// TIA Portal V20 export
ORGANIZATION_BLOCK "Startup"   // OB1005, LAD, Startup
TITLE = "Complete Restart"
// stored: AutoNumber false, Namespace Unit1.Em0, SetENOAutomatically false
   VAR_INPUT
      LostRetentive : Bool;   // True if retentive data are lost
      LostRTC : Bool;   // True if date and time are lost
   END_VAR
BEGIN

REGION Network 1 (SCL): Build the Absolut Reference Designator
   // Set the Absoult Reference Designator in the Config DB
   IF LEN(IN := "Unit1.Em0.Config".em.referenceDesignator.parent) <> 0 THEN
       "Unit1.Em0.Config".em.referenceDesignator.combined := CONCAT_WSTRING(IN1 := "Unit1.Em0.Config".em.referenceDesignator.parent, IN2 := WSTRING#'.', IN3 := "Unit1.Em0.Config".em.referenceDesignator.relative);
   ELSE
       "Unit1.Em0.Config".em.referenceDesignator.combined := "Unit1.Em0.Config".em.referenceDesignator.relative;
   END_IF;
END_REGION

REGION Network 2 (SCL): EM Startup
   "Unit1.Em0.HmiInterface".em.interlinkMode.isLinked := FALSE;
END_REGION

REGION Network 3 (SCL): Assign axes data
   // Assign axes
   "Unit1.Em0.Config".axis[1] := "BA010AZCRDR1_UnwinderLeftAxisB";

   // HW_SubModule
   "Unit1.Em0.Config".moduleAccessPoint[1] := "BA010AZCRCU1~BA010AZCRCU1_X150~BA010AZCRDR1_ModuleAccessPoint";
END_REGION

REGION Network 4 (SCL): EM Startup
   "Unit1.Em0.HmiInterface".em.interlinkMode.isLinked := FALSE;

   // FB Enable
   "Unit1.Em0.HmiInterface".cmUnWinderAxisB.commands.enable := TRUE;
END_REGION

REGION Network 5 (SCL): CM Config
   // Unwinder Axis B
   "Unit1.Em0.Config".cmUnWinderAxisB.referenceDesignator := WSTRING#'Left UnWinder Axis B';
   "Unit1.Em0.Config".cmUnWinderAxisB.disableAlarms := FALSE;
   "Unit1.Em0.Config".cmUnWinderAxisB.masterControlPopUp := TRUE;


   // Air Shaft
   "Unit1.Em0.Config".cmAirShaftOnOff.referenceDesignator := WSTRING#'Left Air Shaft';
   "Unit1.Em0.Config".cmAirShaftOnOff.monitoringLeavingFeedback := T#0MS;
   "Unit1.Em0.Config".cmAirShaftOnOff.monitoringReachingFeedback := T#0MS;
   "Unit1.Em0.Config".cmAirShaftOnOff.monitoringDiscrepancy := T#0ms;
   "Unit1.Em0.Config".cmAirShaftOnOff.setOutputHomeContinuously := TRUE;
   "Unit1.Em0.Config".cmAirShaftOnOff.setOutputWorkContinuously := TRUE;
   "Unit1.Em0.Config".cmAirShaftOnOff.disableHomeCommand := FALSE;
   "Unit1.Em0.Config".cmAirShaftOnOff.disableFeedbackHomePos := TRUE;
   "Unit1.Em0.Config".cmAirShaftOnOff.disableFeedbackWorkPos := TRUE;
   "Unit1.Em0.Config".cmAirShaftOnOff.disableAlarms := FALSE;
   "Unit1.Em0.Config".cmAirShaftOnOff.resetOutputsOnError := FALSE;
   "Unit1.Em0.Config".cmAirShaftOnOff.allwaysWaitOnReachingTime := FALSE;


   // Electrode Expel
   "Unit1.Em0.Config".cmExpelFwdBwd.referenceDesignator := WSTRING#'Left Electrode Expel';
   "Unit1.Em0.Config".cmExpelFwdBwd.monitoringLeavingFeedback := T#5s;
   "Unit1.Em0.Config".cmExpelFwdBwd.monitoringReachingFeedback := T#5s;
   "Unit1.Em0.Config".cmExpelFwdBwd.monitoringDiscrepancy := T#0ms;
   "Unit1.Em0.Config".cmExpelFwdBwd.setOutputHomeContinuously := TRUE;
   "Unit1.Em0.Config".cmExpelFwdBwd.setOutputWorkContinuously := TRUE;
   "Unit1.Em0.Config".cmExpelFwdBwd.disableHomeCommand := FALSE;
   "Unit1.Em0.Config".cmExpelFwdBwd.disableFeedbackHomePos := FALSE;
   "Unit1.Em0.Config".cmExpelFwdBwd.disableFeedbackWorkPos := FALSE;
   "Unit1.Em0.Config".cmExpelFwdBwd.disableAlarms := FALSE;
   "Unit1.Em0.Config".cmExpelFwdBwd.resetOutputsOnError := FALSE;
   "Unit1.Em0.Config".cmExpelFwdBwd.allwaysWaitOnReachingTime := FALSE;


   // Radius Measure
   "Unit1.Em0.Config".cmRadiusMeasureAnalogInput.referenceDesignator := WSTRING#'Left Radius Measure';
   "Unit1.Em0.Config".cmRadiusMeasureAnalogInput.physicalUnit := 'mm';
   "Unit1.Em0.Config".cmRadiusMeasureAnalogInput.isUnipolarSignal := TRUE;
   "Unit1.Em0.Config".cmRadiusMeasureAnalogInput.default := 0;
   "Unit1.Em0.Config".cmRadiusMeasureAnalogInput.limitHigh2 := 10000;
   "Unit1.Em0.Config".cmRadiusMeasureAnalogInput.limitHigh1 := 9000;
   "Unit1.Em0.Config".cmRadiusMeasureAnalogInput.limitLow1 := 40;
   "Unit1.Em0.Config".cmRadiusMeasureAnalogInput.limitLow2 := 30;
   "Unit1.Em0.Config".cmRadiusMeasureAnalogInput.processValueMax := 10000;
   "Unit1.Em0.Config".cmRadiusMeasureAnalogInput.processValueMin := 10;
   "Unit1.Em0.Config".cmRadiusMeasureAnalogInput.scaleAnalogUppPoint := 27648;
   "Unit1.Em0.Config".cmRadiusMeasureAnalogInput.scaleAnalogLowPoint := 0;
   "Unit1.Em0.Config".cmRadiusMeasureAnalogInput.scaleProcessUppPoint := 10000;
   "Unit1.Em0.Config".cmRadiusMeasureAnalogInput.scaleProcessLowPoint := 10;
   "Unit1.Em0.Config".cmRadiusMeasureAnalogInput.disableAlarms := FALSE;


   // EPC
   "Unit1.Em0.Config".cmEpc.referenceDesignator := WSTRING#'Left Uniwnder EPC';
   "Unit1.Em0.Config".cmEpc.hwID.EkrOut_Auto_Sp_Acp_HW_ID := "BA010AZCREPCC1~EkrOut_Auto_Sp_Acp_1";
   "Unit1.Em0.Config".cmEpc.hwID.EkrOut_CAM_Data_HW_ID := "BA010AZCREPCC1~EkrOut_CAM_Data_1";
   "Unit1.Em0.Config".cmEpc.hwID.EkrOut_CLS_Data_HW_ID := "BA010AZCREPCC1~EkrOut_CLS_Data_1";
   "Unit1.Em0.Config".cmEpc.hwID.EkrOut_Guiding_edges_HW_ID := "BA010AZCREPCC1~EkrOut_Guiding_edges_1";
   "Unit1.Em0.Config".cmEpc.hwID.EkrOut_HEADER_Data_HW_ID := "BA010AZCREPCC1~EkrOut_HEADER_Data_1";
   "Unit1.Em0.Config".cmEpc.hwID.EkrOut_POS_unit_HW_ID := "BA010AZCREPCC1~EkrOut_POS_unit_1";
   "Unit1.Em0.Config".cmEpc.hwID.EkrOut_SEN_Data_HW_ID := "BA010AZCREPCC1~EkrOut_SEN_Data_1";
   "Unit1.Em0.Config".cmEpc.hwID.EkrOut_Servo_Center_HW_ID := "BA010AZCREPCC1~EkrOut_Servo_Center_1";
   "Unit1.Em0.Config".cmEpc.hwID.EkrOut_Setpoint_HW_ID := "BA010AZCREPCC1~EkrOut_Setpoint_1";
   "Unit1.Em0.Config".cmEpc.hwID.EkrOut_Web_width_HW_ID := "BA010AZCREPCC1~EkrOut_Web_width_1";
   "Unit1.Em0.Config".cmEpc.hwID.EkrIn_Auto_Sp_Acp_HW_ID := "BA010AZCREPCC1~EkrIn_Auto_Sp_Acp_1";
   "Unit1.Em0.Config".cmEpc.hwID.EkrIn_HEADER_Data_HW_ID := "BA010AZCREPCC1~EkrIn_HEADER_Data_1";
   "Unit1.Em0.Config".cmEpc.hwID.EkrIn_POS_unit_HW_ID := "BA010AZCREPCC1~EkrIn_POS_unit_1";
   "Unit1.Em0.Config".cmEpc.hwID.EkrIn_Setpoint_HW_ID := "BA010AZCREPCC1~EkrIn_Setpoint_1";
   "Unit1.Em0.Config".cmEpc.hwID.EkrIn_Web_width_HW_ID := "BA010AZCREPCC1~EkrIn_Web_width_1";


   // Tension Check Sensor
   "Unit1.Em0.Config".cmTensionCheckSensor.referenceDesignator := WSTRING#'DigitalSignal';
   "Unit1.Em0.Config".cmTensionCheckSensor.onDelay := T#0ms;
   "Unit1.Em0.Config".cmTensionCheckSensor.offDelay := T#0ms;
   "Unit1.Em0.Config".cmTensionCheckSensor.default := false;
   "Unit1.Em0.Config".cmTensionCheckSensor.invertProcessValue := false;
   "Unit1.Em0.Config".cmTensionCheckSensor.disableAlarms := false;


   // Radius Measure AddOn
   // Config.cmRadiusMeasure.Offset := HmiInterface.cmRadiusMeasure.configuration.Offset := 91.0;//제로셋 세팅시 직경
   // Config.cmRadiusMeasure.DecimalPoint := HmiInterface.cmRadiusMeasure.configuration.DecimalPoint := 1;
   "Unit1.Em0.Config".cmRadiusMeasure.Offset := "Unit1.Em0.HmiInterface".cmRadiusMeasure.configuration.Offset := 70.0;//제로셋 세팅시 반경 -> 원익한테 받아서 정밀값 세팅하면됨 
   "Unit1.Em0.Config".cmRadiusMeasure.DecimalPoint := "Unit1.Em0.HmiInterface".cmRadiusMeasure.configuration.DecimalPoint := 1;
END_REGION
END_ORGANIZATION_BLOCK
